// TIA Portal V20 export
FUNCTION_BLOCK "Fx_LadEdges"   // FB3, LAD
{ S7_Optimized_Access := 'TRUE' }
// stored: MemoryReserve 100, SetENOAutomatically false
   VAR_INPUT
      "a" : Bool;
      "b" : Bool;
      c : Bool;
   END_VAR
   VAR_OUTPUT
      pe : Bool;
      ne : Bool;
      pc : Bool;
      nc : Bool;
      trig : Bool;
      notOut : Bool;
      inv : Bool;
      orOut : Bool;
      split1 : Bool;
      split2 : Bool;
      latch1 : Bool;
      latch2 : Bool;
      held : Bool;
   END_VAR
   VAR
      m1 : Bool;
      m2 : Bool;
      m3 : Bool;
      m4 : Bool;
      m5 : Bool;
      sr : Bool;
      rs : Bool;
   END_VAR
   VAR_TEMP   // added for the SCL form of the ladder/FBD networks
      _w1 : Bool;
   END_VAR
BEGIN

REGION Network 1
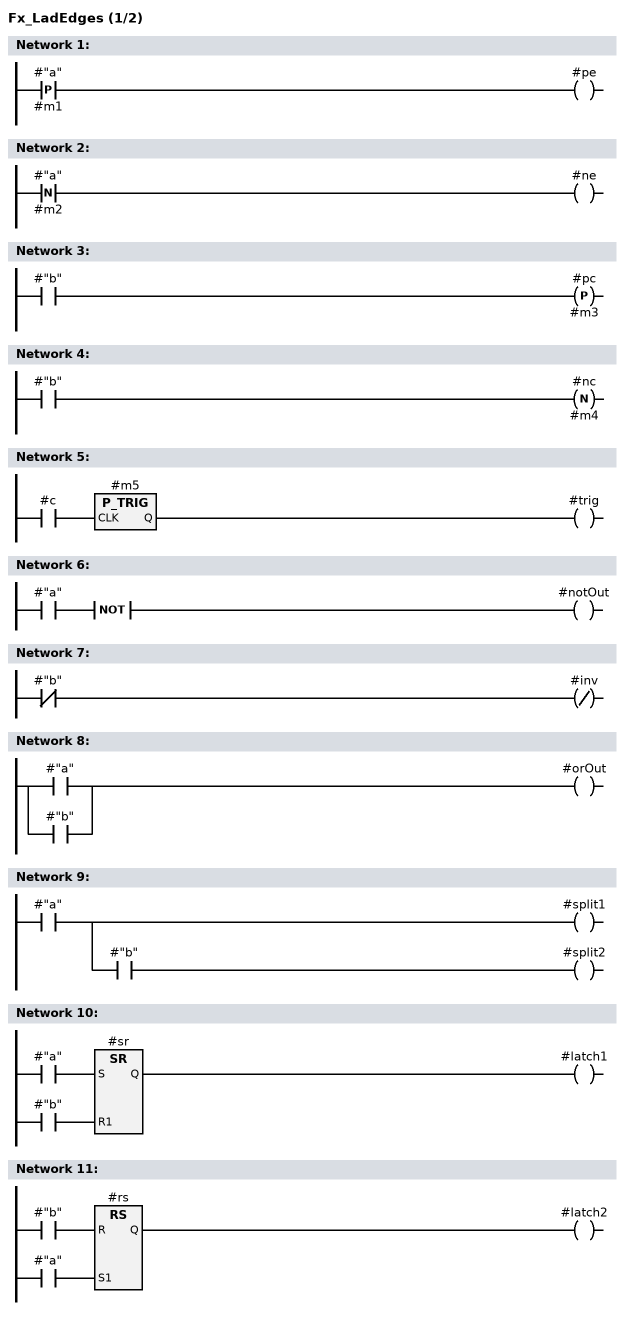
   RUNG wire#powerrail
      P_Contact(operand := #"a", bit := #m1)
      Coil( #pe )
   END_RUNG
   // the same network as SCL:
   #_w1 := #"a" AND NOT #m1;   // rising edge of #"a"
   #m1 := #"a";
   #pe := #_w1;
END_REGION

REGION Network 2
   RUNG wire#powerrail
      N_Contact(operand := #"a", bit := #m2)
      Coil( #ne )
   END_RUNG
   // the same network as SCL:
   #_w1 := NOT #"a" AND #m2;   // falling edge of #"a"
   #m2 := #"a";
   #ne := #_w1;
END_REGION

REGION Network 3
   #pc := #"b" AND NOT #m3;   // rising edge
   #m3 := #"b";
END_REGION

REGION Network 4
   #nc := NOT #"b" AND #m4;   // falling edge
   #m4 := #"b";
END_REGION

REGION Network 5
   RUNG wire#powerrail
      Contact( #c )
      P_Trig( #m5 )
      Coil( #trig )
   END_RUNG
   // the same network as SCL:
   #_w1 := #c AND NOT #m5;   // rising edge
   #m5 := #c;
   #trig := #_w1;
END_REGION

REGION Network 6
   RUNG wire#powerrail
      Contact( #"a" )
      Not()
      Coil( #notOut )
   END_RUNG
   // the same network as SCL:
   #notOut := NOT #"a";
END_REGION

REGION Network 7
   RUNG wire#powerrail
      I_Contact( #"b" )
      I_Coil( #inv )
   END_RUNG
   // the same network as SCL:
   #inv := NOT (NOT #"b");
END_REGION

REGION Network 8
   RUNG wire#powerrail
      Contact( #"a" )
      wire#w1
      Coil( #orOut )
   END_RUNG
   RUNG wire#powerrail
      Contact( #"b" )
   END_RUNG wire#w1
   // the same network as SCL:
   #orOut := #"a" OR #"b";
END_REGION

REGION Network 9
   RUNG wire#powerrail
      Contact( #"a" )
      wire#w1
      Coil( #split1 )
   END_RUNG
   RUNG wire#w1
      Contact( #"b" )
      Coil( #split2 )
   END_RUNG
   // the same network as SCL:
   #split1 := #"a";
   #split2 := #"a" AND #"b";
END_REGION

REGION Network 10
   RUNG wire#powerrail
      Contact( #"a" )
      S_SR(operand := #sr, r1 := wire#w1)
      Coil( #latch1 )
   END_RUNG
   RUNG wire#powerrail
      Contact( #"b" )
   END_RUNG wire#w1
   // the same network as SCL:
   IF #"a" THEN
       #sr := TRUE;   // SR flip-flop
   END_IF;
   IF #"b" THEN #sr := FALSE; END_IF;
   #latch1 := #sr;
END_REGION

REGION Network 11
   RUNG wire#powerrail
      Contact( #"b" )
      S_RS(operand := #rs, s1 := wire#w1)
      Coil( #latch2 )
   END_RUNG
   RUNG wire#powerrail
      Contact( #"a" )
   END_RUNG wire#w1
   // the same network as SCL:
   IF #"b" THEN
       #rs := FALSE;   // RS flip-flop
   END_IF;
   IF #"a" THEN #rs := TRUE; END_IF;
   #latch2 := #rs;
END_REGION

REGION Network 12
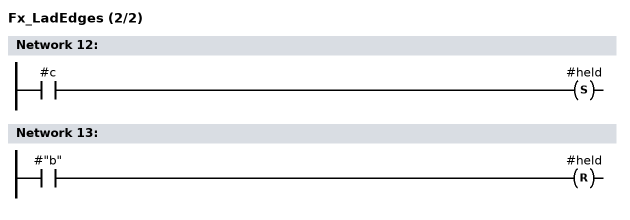
   RUNG wire#powerrail
      Contact( #c )
      S_Coil( #held )
   END_RUNG
   // the same network as SCL:
   IF #c THEN #held := TRUE; END_IF;
END_REGION

REGION Network 13
   RUNG wire#powerrail
      Contact( #"b" )
      R_Coil( #held )
   END_RUNG
   // the same network as SCL:
   IF #"b" THEN #held := FALSE; END_IF;
END_REGION
END_FUNCTION_BLOCK
